Fanuc KAREL source: CA0050.KL

PROGRAM CA0050
%STACKSIZE=65535
%PRIORITY=65535
%NOLOCKGROUP
TYPE
T=STRUCTURE
A : INTEGER
B : REAL
ENDSTRUCTURE
VAR
G : INTEGER
I : INTEGER
R : REAL
B : BOOLEAN
S : STRING[16]
AI : ARRAY[2] OF INTEGER
AR : ARRAY[2] OF REAL
ST : T
P : XYZWPR
V : VECTOR
ROUTINE F(P1 : INTEGER; P2 : REAL; P3 : BOOLEAN; P4 : STRING; P5 : INTEGER; P6 : REAL; P7 : BOOLEAN; P8 : STRING; P9 : INTEGER; P10 : REAL; P11 : BOOLEAN; P12 : STRING; P13 : INTEGER; P14 : REAL; P15 : BOOLEAN; P16 : STRING; P17 : INTEGER;
P18 : REAL; P19 : BOOLEAN; P20 : STRING; P21 : INTEGER; P22 : REAL; P23 : BOOLEAN; P24 : STRING; P25 : INTEGER; P26 : REAL; P27 : BOOLEAN; P28 : STRING; P29 : INTEGER; P30 : REAL; P31 : BOOLEAN; P32 : STRING) FROM CA0050
ROUTINE F
BEGIN
G=(G + 1)
END F
BEGIN
G=0
I=1
R=2.5
B=TRUE
S='A'
AI[1]=3
AR[1]=4.5
-- UNSAFE_SOURCE_IR line 62: ST.A = 5
-- UNSAFE_SOURCE_IR line 63: ST.B = 6.5
F(I,R,B,S,I,R,B,S,I,R,B,S,I,R,B,S,I,R,B,S,I,R,B,S,I,R,B,S,I,R,B,S)
END CA0050
